INTERFACE ITF_BaseComponent EXTENDS ITF_BaseLoggerElement

(*			
	RafalOS
	Rafał Osajda		27.03.2025		TC 4024.66
	Obsluga bledow sprawdzanie czy jakis blad sie nei pojawil i ustawienie stanu lub wylaczenie
*)
METHOD PUBLIC ExecuteEveryCycle_Error
VAR_INPUT
END_VAR
END_METHOD

(*			
	RafalOS
	Rafał Osajda		27.03.2025		TC 4024.66
	Wywolanie co cykl operacji 
*)
METHOD PUBLIC ExecuteEveryCycle_Operation
VAR_INPUT
END_VAR
END_METHOD

(*			
	RafalOS
	Rafał Osajda		27.03.2025		TC 4024.66
	Aktualizacja flag 
*)
METHOD PUBLIC ExecuteEveryCycle_Status
VAR_INST
END_VAR
END_METHOD

(*			
	RafalOS
	Rafał Osajda		27.03.2025		TC 4024.66
	Testowanie czy nei pojawil sie jakis rozkaz i uruchomienie odpowiednich operacji
*)
METHOD PUBLIC ExecuteEveryCycle_Test
VAR_INPUT
END_VAR
END_METHOD

METHOD PUBLIC FirstCycle : BOOL
VAR_INPUT
END_VAR
END_METHOD

METHOD PUBLIC IsValidCommonData : BOOL
VAR_INPUT
END_VAR
END_METHOD

(*			
	RafalOS
	Rafał Osajda		07.10.2025		TC 4024.66
	Dodpisywanie się do listy logera
*)
METHOD PUBLIC JoinTheLogger : BOOL
VAR_INPUT
END_VAR
END_METHOD

METHOD PUBLIC LinkCommonData : BOOL
VAR_INPUT
	stCommonData				: REFERENCE TO ST_BaseCommonData;
END_VAR
END_METHOD

(*			
	RafalOS
	Rafał Osajda		26.03.2025		TC 4024.66
	Dodawanie parametru do elementu wykonawczego - metode wywołać przy pierwszym uruchomieniu programu by wgrać parametry do pamięci
	później używać tylko edycji lub przywracania wartości domyślnych
*)
METHOD PUBLIC ParameterAdd : BOOL
VAR_INPUT
	stParameter			: ST_BaseDescriptor;
END_VAR
END_METHOD

(*			
	RafalOS
	Rafał Osajda		26.03.2025		TC 4024.66
	Modyfikuje wartość domyślną w istniejącym parametrze - true jak się zmiana udała
*)
METHOD PUBLIC ParameterCorrectDefaultValue : BOOL
VAR_INPUT
	uiNumber			: UINT;
	rValue				: REAL;
END_VAR
END_METHOD

METHOD PUBLIC ParameterCorrectName : BOOL
VAR_INPUT
	eLocation					: E_BaseLocation;
	uiNumberOfParameter			: UINT;
	wsDescription				: WSTRING;
END_VAR
END_METHOD

(*			
	RafalOS
	Rafał Osajda		26.03.2025		TC 4024.66
	Modyfikuje wartość w istniejącym parametrze - true jak się zmiana udała
*)
METHOD PUBLIC ParameterCorrectValue : BOOL
VAR_INPUT
	uiNumber			: UINT;
	rValue				: REAL;
END_VAR
END_METHOD

METHOD PUBLIC ParameterGet : ST_BaseDescriptor
VAR_INPUT
	uiNumer				: UINT;
END_VAR
END_METHOD

(*			
	RafalOS
	Rafał Osajda		26.03.2025		TC 4024.66
	Zwraca wartosc domyslna
*)
METHOD PUBLIC ParameterGetDefaultValue : REAL
VAR_INPUT
	uiNumber				: UINT;
END_VAR
END_METHOD

(*			
	RafalOS
	Rafał Osajda		26.03.2025		TC 4024.66
	Zwraca wartość MAX
*)
METHOD PUBLIC ParameterGetMax : REAL
VAR_INPUT
	uiNumber				: UINT;
END_VAR
END_METHOD

(*			
	RafalOS
	Rafał Osajda		26.03.2025		TC 4024.66
	Zwraca wartość MIN
*)
METHOD PUBLIC ParameterGetMin : REAL
VAR_INPUT
	uiNumber				: UINT;
END_VAR
END_METHOD

METHOD PUBLIC ParameterGetNumberOfAdded : UINT
VAR_INPUT
END_VAR
END_METHOD

(*			
	RafalOS
	Rafał Osajda		26.03.2025		TC 4024.66
	Zwraca jednostke
*)
METHOD PUBLIC ParameterGetUnit : STRING(6)
VAR_INPUT
	uiNumber				: uINT;
END_VAR
END_METHOD

(*			
	RafalOS
	Rafał Osajda		26.03.2025		TC 4024.66
	Zwraca wartość
*)
METHOD PUBLIC ParameterGetValue : REAL
VAR_INPUT
	uiNumber				: UINT;
END_VAR
END_METHOD

(*			
	RafalOS
	Rafał Osajda		26.03.2025		TC 4024.66
	Modyfikacja istniejącego parametra jako przypisanie nowego deskryptora
*)
METHOD PUBLIC ParameterModify : BOOL
VAR_INPUT
	uiNumber			: UINT;
	stParameter			: ST_BaseDescriptor;
END_VAR
END_METHOD

METHOD PUBLIC ParameterRestoreDefaultValue : BOOL
VAR_INPUT
	uiNumber		: UINT;
END_VAR
END_METHOD

(*			
	RafalOS
	Rafał Osajda		04.05.2025		TC 4024.66
	Skasowanie i utworzenie tablicy parametrów od nowa 
*)
METHOD PUBLIC ParametersCreate : BOOL
END_METHOD

(*			
	RafalOS
	Rafał Osajda		04.05.2025		TC 4024.66
	Przywrocenie parametrow - in na false to tylko ten element true razem z podelementami
*)
METHOD PUBLIC ParameterSetToDefault : BOOL
END_METHOD

METHOD PUBLIC Reset : BOOL
VAR_INPUT
END_VAR
END_METHOD

METHOD PUBLIC ResetGetBusy : BOOL
VAR_INPUT
END_VAR
END_METHOD

METHOD PUBLIC ResetGetStatus : BOOL
VAR_INPUT
END_VAR
END_METHOD

END_INTERFACE

(* stored: Version 1.1.0.1
   Itf ITF_BaseComponent: Id {bfd259ad-b5a7-0c3e-25af-f416d786cc1f}
   Folder Parameter: Id {162355fc-3282-0c2e-2d48-030ede6ecd3a}
   Method ExecuteEveryCycle_Error: Id {9687ff7f-0d6e-0d51-23a3-336377b58d2c}
   Method ExecuteEveryCycle_Operation: Id {84e8e489-e3ad-03cb-399e-9ce5e19542d8}
   Method ExecuteEveryCycle_Status: Id {a817f84c-463c-04f3-0e77-c3fd90132b64}
   Method ExecuteEveryCycle_Test: Id {9b8a596a-c333-0a36-2211-eb0d1ec8eb39}
   Method FirstCycle: Id {5bb3c28d-6dff-0c9d-3483-ca1fcada3e23}
   Method IsValidCommonData: Id {79422fac-c686-0f81-2652-4e5411a92a86}
   Method JoinTheLogger: Id {6452dc54-6621-0a82-3e77-69f38e77752f}
   Method LinkCommonData: Id {a28b3732-9a1a-0508-12b7-66129c063dab}
   Method ParameterAdd: Id {cb2832e6-b124-0d0c-38c6-780ac9f7fc1b}
   Method ParameterCorrectDefaultValue: Id {4bbe970d-6672-018d-1d17-344ff0ac718a}
   Method ParameterCorrectName: Id {6ec96585-99ee-0c3d-1ca5-f52d44d2781a}
   Method ParameterCorrectValue: Id {5c025912-789a-0744-1c53-d16d2837f884}
   Method ParameterGet: Id {21d37c06-febc-07f0-1a30-ea03aba0338c}
   Method ParameterGetDefaultValue: Id {4f87981f-6989-0e65-1fcf-fb3647acf1ca}
   Method ParameterGetMax: Id {4b75e398-c9ba-09cb-0312-dd60c23d0d65}
   Method ParameterGetMin: Id {6889c42b-5d50-0a09-0e6b-5ce55ebd8346}
   Method ParameterGetNumberOfAdded: Id {54c667d7-5f5e-0690-1dc5-6970b5099c23}
   Method ParameterGetUnit: Id {a76199e2-2fb6-08b3-12ae-6d01fe05455e}
   Method ParameterGetValue: Id {9424063b-795d-0b64-3fc5-8cce9ff5d1eb}
   Method ParameterModify: Id {8f713bac-a4fa-07d4-0764-9b59380d937d}
   Method ParameterRestoreDefaultValue: Id {030f6759-bd3d-00b9-02b0-bd91925d754f}
   Method ParametersCreate: Id {f87dac04-0e60-0cf9-3fcb-2ab850eac29d}
   Method ParameterSetToDefault: Id {76330915-de2f-01b9-34f0-39db59d2b98e}
   Method Reset: Id {77eb7b91-893b-0d84-16a4-ac22c2bb7b56}
   Method ResetGetBusy: Id {889fd0ad-7a78-0e51-0d48-1f63919c6997}
   Method ResetGetStatus: Id {494afb3a-3397-0df4-0cc3-a3d06f85b5a6} *)
